{attribute 'qualified_only'}
VAR_GLOBAL
	ECnv_Sys:  ARRAY[1..2] OF ECnv_Control_DUT;
	LCnv_Sys:  ARRAY[1..2] OF Cnv_VTD_Control_DUT;
	VTD_Sys:  ARRAY[1..2] OF VTD_Control_DUT;
	VTD_Order_Table:  ARRAY[1..2] OF WMS_OPC_UA_DUT;
	Buffer_Order_Table:  ARRAY[1..2] OF WMS_OPC_UA_DUT;
// 	Shuttles_Position:  ARRAY[1..10] OF STRUCT;
	VTDBarcode_Station:  ARRAY[1..2] OF Barcode_Station_DUT;
	Gate_Station:  ARRAY[1..3] OF Gate_Station_DUT;
	Charger_Level:  ARRAY[2..6] OF Charger_DUT;
// 	Movement_Completed:  STRUCT;
END_VAR

(* stored: Version 1.1.0.1
   GVL Control: Id {5e6952d4-e20c-4a7f-aad7-0649e4f09d9f} *)
